FUNCTION_BLOCK FB_Base_Stack IMPLEMENTS I_Stack
VAR_INPUT
END_VAR
VAR_OUTPUT
END_VAR
VAR
END_VAR

{warning 'add method implementation '}
METHOD Peek : T_DATA_TYPE
END_METHOD

{warning 'add method implementation '}
METHOD Pop
END_METHOD

{warning 'add method implementation '}
METHOD Push
VAR_INPUT
	Data	: T_DATA_TYPE;
END_VAR
END_METHOD

{warning 'add method implementation '}
METHOD Show
END_METHOD

END_FUNCTION_BLOCK

(* stored: Version 1.1.0.1, ProductVersion 3.1.4024.4
   POU FB_Base_Stack: Id {8bc58612-cbbe-4e93-b171-775069cb599d}, SpecialFunc None
   Method Peek: Id {172dc61e-e2a8-48a9-ae38-b6a973d240ec}
   Method Pop: Id {f233d5b4-3108-4337-b281-dc937455ad33}
   Method Push: Id {354dceed-21d1-48bb-bcb2-2026d0a92934}
   Method Show: Id {6e723a8f-bd16-42eb-9cf9-40357cb7d068} *)
